FUNCTION CEIL : INT
VAR_INPUT
	X : REAL;
END_VAR


(*
version 1.1	21. mar. 2008
programmer 	hugo
tested by	tobias

This is a rounding function which returns the smallest possible integer which is greater or equal to X.
ceil(3.14) = 4
ceil(-3.14) = -3

*)

CEIL := REAL_TO_INT(x);
IF CEIL < X THEN
	CEIL := CEIL + 1;
END_IF;


(* revision history
hm	7. feb. 2007	rev 1.0
	original version

hm	21. mar. 2008	rev 1.1
	use REAL_TO_INT instead of trunc for compatibility reasons

*)

END_FUNCTION

(* stored: Version 1.1.0.1, ProductVersion 3.1.4022.7
   POU CEIL: Id {1a4b2aab-c597-44bc-b129-b360db84ba94}, SpecialFunc None *)
